// TIA Portal project "Takt_Docas_V13_SP1_V15" (V15)
// Software para a implementação do  Takt nas docas da fábrica do "KD".

(* hardware
DEVICE "S7-1200 station_1"  S7-1200 Station
   slot 0: "Rack_0"  Rack  V1.0
   slot 1: "PLC_Docas"  CPU 1214C DC/DC/DC  6ES7 214-1AG40-0XB0  V4.0
*)

// ===== PLC "PLC_Docas"  CPU 1214C DC/DC/DC =====

VAR_GLOBAL   // PLC tag table "Default tag table"
   "System_Byte" AT %MB1 : Byte;
   "FirstScan" AT %M1.0 : Bool;
   "DiagStatusUpdate" AT %M1.1 : Bool;
   "AlwaysTRUE" AT %M1.2 : Bool;
   "AlwaysFALSE" AT %M1.3 : Bool;
   "Clock_Byte" AT %MB0 : Byte;
   "Clock_10Hz" AT %M0.0 : Bool;
   "Clock_5Hz" AT %M0.1 : Bool;
   "Clock_2.5Hz" AT %M0.2 : Bool;
   "Clock_2Hz" AT %M0.3 : Bool;
   "Clock_1.25Hz" AT %M0.4 : Bool;
   "Clock_1Hz" AT %M0.5 : Bool;
   "Clock_0.625Hz" AT %M0.6 : Bool;
   "Clock_0.5Hz" AT %M0.7 : Bool;
   "Tag_1" AT %M100.0 : Bool;
   "startsystem" AT %I1.0 : Bool;
END_VAR

VAR_GLOBAL   // PLC tag table "Peripheral_inputs"
   "P.IN_Reset_Andon_doca1" AT %I0.0 : Bool;   // Entrada pereférica para resetar a chamada de Andon da "doca 1"
   "P.IN_Andon_doca1" AT %I0.1 : Bool;   // Entrada pereférica para chamada de Andon "doca 1"
   "P.IN_Reset_Andon_doca2" AT %I0.2 : Bool;   // Entrada pereférica para resetar a chamada de Andon da "doca 2"
   "P.IN_Andon_doca2" AT %I0.3 : Bool;   // Entrada pereférica para chamada de Andon "doca 2"
   "P.IN_Reset_Andon_doca3" AT %I0.4 : Bool;   // Entrada pereférica para resetar a chamada de Andon da "doca 3"
   "P.IN_Andon_doca3" AT %I0.5 : Bool;   // Entrada pereférica para chamada de Andon "doca 3"
   "P.IN_Reset_Andon_doca4" AT %I0.6 : Bool;   // Entrada pereférica para resetar a chamada de Andon da "doca 4"
   "P.IN_Andon_doca4" AT %I0.7 : Bool;   // Entrada pereférica para chamada de Andon "doca 4"
END_VAR

// folder: DBs

DATA_BLOCK "Input_memory"   // DB1
{ S7_Optimized_Access := 'TRUE' }
VERSION : 0.1
   VAR
      "M.S_IN_Reset_Andon_doca1" : Bool;   // Memória de movimentação do sinal de entrada do reset da chamada de Andon "doca1".
      "M.S_IN_Andon_doca1" : Bool;   // Memória de movimentação do sinal de entrada para chamada de andon "doca1".
      "M.S_IN_Reset_Andon_doca2" : Bool;   // Memória de movimentação do sinal de entrada do reset da chamada de Andon "doca2".
      "M.S_IN_Andon_doca2" : Bool;   // Memória de movimentação do sinal de entrada para chamada de andon "doca2".
      "M.S_IN_Reset_Andon_doca3" : Bool;   // Memória de movimentação do sinal de entrada do reset da chamada de Andon "doca3".
      "M.S_IN_Andon_doca3" : Bool;   // Memória de movimentação do sinal de entrada para chamada de andon "doca3".
      "M.S_IN_Reset_Andon_doca4" : Bool;   // Memória de movimentação do sinal de entrada do reset da chamada de Andon "doca4".
      "M.S_IN_Andon_doca4" : Bool;   // Memória de movimentação do sinal de entrada para chamada de andon "doca4".
   END_VAR
BEGIN
END_DATA_BLOCK

DATA_BLOCK "Output_memory"   // DB2
{ S7_Optimized_Access := 'TRUE' }
VERSION : 0.1
BEGIN
END_DATA_BLOCK

// folder: DBs_FBs

DATA_BLOCK "FB500_Dock_Takt_DB"   // DB3
{ S7_Optimized_Access := 'FALSE' }
VERSION : 0.1
// stored: InstanceOfName FB500_Dock_Takt
"FB500_Dock_Takt"
BEGIN
END_DATA_BLOCK

DATA_BLOCK "FB500_Dock_Takt_DB_1"   // DB4
{ S7_Optimized_Access := 'FALSE' }
VERSION : 0.1
// stored: InstanceOfName FB500_Dock_Takt
"FB500_Dock_Takt"
BEGIN
END_DATA_BLOCK

DATA_BLOCK "FB500_Dock_Takt_DB_2"   // DB5
{ S7_Optimized_Access := 'FALSE' }
VERSION : 0.1
// stored: InstanceOfName FB500_Dock_Takt
"FB500_Dock_Takt"
BEGIN
END_DATA_BLOCK

DATA_BLOCK "FB500_Dock_Takt_DB_3"   // DB6
{ S7_Optimized_Access := 'FALSE' }
VERSION : 0.1
// stored: InstanceOfName FB500_Dock_Takt
"FB500_Dock_Takt"
BEGIN
END_DATA_BLOCK

DATA_BLOCK "stopstar_DB"   // DB9
{ S7_Optimized_Access := 'TRUE' }
VERSION : 0.1
// stored: InstanceOfName Andon_Call
"Andon_Call"
BEGIN
END_DATA_BLOCK

// folder: DBs_System

DATA_BLOCK "Inputs_memory.system"   // DB7
{ S7_Optimized_Access := 'FALSE' }
VERSION : 0.1
   VAR
      "M.S_IN_Timer.Takt.D1" : Time;   // Memória de leitura do Sistema para parâmetrizar o tempo do Takt na "doca 1".
      "M.S_IN_Dock_goal.D1" : Int;   // Memória de leitura do Sistema para parâmetrizar o objetivo de produção na "doca 1".
      "M.S_IN_Timer.Takt.D2" : Time;   // Memória de leitura do Sistema para parâmetrizar o tempo do Takt na "doca 2".
      "M.S_IN_Dock_goal.D2" : Int;   // Memória de leitura do Sistema para parâmetrizar o objetivo de produção na "doca 2".
      "M.S_IN_Timer.Takt.D3" : Time;   // Memória de leitura do Sistema para parâmetrizar o tempo do Takt na "doca 3".
      "M.S_IN_Dock_goal.D3" : Int;   // Memória de leitura do Sistema para parâmetrizar o objetivo de produção na "doca 3".
      "M.S_IN_Timer.Takt.D4" : Time;   // Memória de leitura do Sistema para parâmetrizar o tempo do Takt na "doca 4".
      "M.S_IN_Dock_goal.D4" : Int;   // Memória de leitura do Sistema para parâmetrizar o objetivo de produção na "doca 4".
      "M.S_IN_Enable.Takt" : Bool;   // Memória de leitura do Sistema para habilitar o Takt das docas.
      StartBySystem1 : Bool;
      StartBySystem2 : Bool;
      StartBySystem3 : Bool;
      StartBySystem4 : Bool;
      Empty5 : Bool;
      Empty6 : Bool;
      Empty7 : Bool;
   END_VAR
BEGIN
END_DATA_BLOCK

DATA_BLOCK "Outputs_memory.system"   // DB8
{ S7_Optimized_Access := 'FALSE' }
VERSION : 0.1
   VAR
      "M.S_Out_TaktActual.D1" : Time;   // Memória de leitura do Sistema com o valor do Takt atual da "doca 1".
      "M.S_Out_StopTime.D1" : Time;   // Memória de leitura do Sistema com o valor do Stop time da "doca 1".
      "M.S_Out_Production.D1" : Int;   // Memória de leitura do Sistema com o valor da Produção até o momento da "doca 1"
      "M.S_Out_Dock_goal.D1" : Int;   // Memória de leitura do Sistema com o valor do objetivo de produção da "doca 1"
      "M.S_Out_TaktActual.D2" : Time;   // Memória de leitura do Sistema com o valor do Takt atual da "doca 2".
      "M.S_Out_StopTime.D2" : Time;   // Memória de leitura do Sistema com o valor do Stop time da "doca 2".
      "M.S_Out_Production.D2" : Int;   // Memória de leitura do Sistema com o valor da Produção até o momento da "doca 2"
      "M.S_Out_Dock_goal.D2" : Int;   // Memória de leitura do Sistema com o valor do objetivo de produção da "doca 2"
      "M.S_Out_TaktActual.D3" : Time;   // Memória de leitura do Sistema com o valor do Takt atual da "doca 3".
      "M.S_Out_StopTime.D3" : Time;   // Memória de leitura do Sistema com o valor do Stop time da "doca 3".
      "M.S_Out_Production.D3" : Int;   // Memória de leitura do Sistema com o valor da Produção até o momento da "doca 3"
      "M.S_Out_Dock_goal.D3" : Int;   // Memória de leitura do Sistema com o valor do objetivo de produção da "doca 3"
      "M.S_Out_TaktActual.D4" : Time;   // Memória de leitura do Sistema com o valor do Takt atual da "doca 4".
      "M.S_Out_StopTime.D4" : Time;   // Memória de leitura do Sistema com o valor do Stop time da "doca 4".
      "M.S_Out_Production.D4" : Int;   // Memória de leitura do Sistema com o valor da Produção até o momento da "doca 4"
      "M.S_Out_Dock_goal.D4" : Int;   // Memória de leitura do Sistema com o valor do objetivo de produção da "doca 4"
      "M.S_Out_Stuffing_target" : Int;   // Memória de leitura do Sistema com o valor do objetivo diario total da estufagem.
      "M.S_Out_Andon.D1" : Bool;   // Memória de leitura do Sistema da chamada de Andon da "doca 1".
      "M.S_Out_Andon.D2" : Bool;   // Memória de leitura do Sistema da chamada de Andon da "doca 2".
      "M.S_Out_Andon.D3" : Bool;   // Memória de leitura do Sistema da chamada de Andon da "doca 3".
      "M.S_Out_Andon.D4" : Bool;   // Memória de leitura do Sistema da chamada de Andon da "doca 4".
      Empty : Bool;
      Empty_1 : Bool;
      Empty_2 : Bool;
      Empty_3 : Bool;
   END_VAR
BEGIN
END_DATA_BLOCK

// folder: (top level)

ORGANIZATION_BLOCK "Main"   // OB1, LAD, ProgramCycle
TITLE = "Main Program Sweep (Cycle)"
{ S7_Optimized_Access := 'TRUE' }
VERSION : 0.1
   VAR_INPUT
      Initial_Call : Bool;   // Initial call of this OB
      Remanence : Bool;   // =True, if remanent data are available
   END_VAR
BEGIN

REGION Network 1: Peripheral Signals (Andon_Call)
   // Movimentação dos sinais das entradas periféricas para as memórias de movimentação.
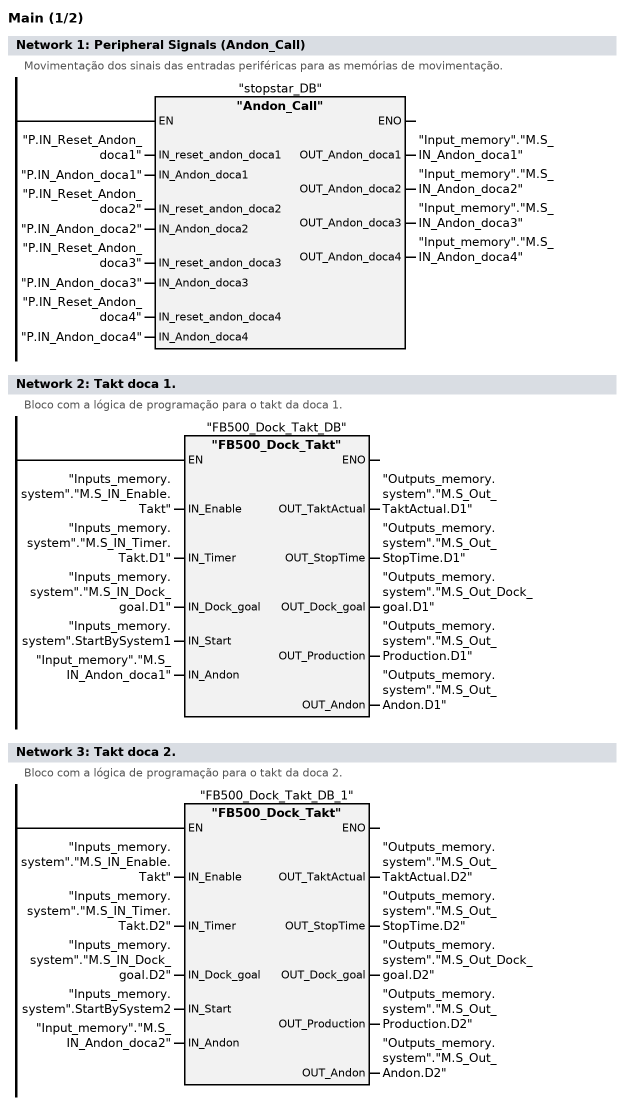
   RUNG wire#powerrail
      "stopstar_DB"(IN_reset_andon_doca1 := "P.IN_Reset_Andon_doca1", IN_Andon_doca1 := "P.IN_Andon_doca1", IN_reset_andon_doca2 := "P.IN_Reset_Andon_doca2", IN_Andon_doca2 := "P.IN_Andon_doca2", IN_reset_andon_doca3 := "P.IN_Reset_Andon_doca3", IN_Andon_doca3 := "P.IN_Andon_doca3", IN_reset_andon_doca4 := "P.IN_Reset_Andon_doca4", IN_Andon_doca4 := "P.IN_Andon_doca4", OUT_Andon_doca1 => "Input_memory"."M.S_IN_Andon_doca1", OUT_Andon_doca2 => "Input_memory"."M.S_IN_Andon_doca2", OUT_Andon_doca3 => "Input_memory"."M.S_IN_Andon_doca3", OUT_Andon_doca4 => "Input_memory"."M.S_IN_Andon_doca4")
   END_RUNG
   // the same network as SCL:
   "stopstar_DB"(IN_reset_andon_doca1 := "P.IN_Reset_Andon_doca1",   // "Andon_Call"
                 IN_Andon_doca1 := "P.IN_Andon_doca1",
                 IN_reset_andon_doca2 := "P.IN_Reset_Andon_doca2",
                 IN_Andon_doca2 := "P.IN_Andon_doca2",
                 IN_reset_andon_doca3 := "P.IN_Reset_Andon_doca3",
                 IN_Andon_doca3 := "P.IN_Andon_doca3",
                 IN_reset_andon_doca4 := "P.IN_Reset_Andon_doca4",
                 IN_Andon_doca4 := "P.IN_Andon_doca4",
                 OUT_Andon_doca1 => "Input_memory"."M.S_IN_Andon_doca1",
                 OUT_Andon_doca2 => "Input_memory"."M.S_IN_Andon_doca2",
                 OUT_Andon_doca3 => "Input_memory"."M.S_IN_Andon_doca3",
                 OUT_Andon_doca4 => "Input_memory"."M.S_IN_Andon_doca4");
END_REGION

REGION Network 2: Takt doca 1.
   // Bloco com a lógica de programação para o takt da doca 1.
   RUNG wire#powerrail
      "FB500_Dock_Takt_DB"(IN_Enable := "Inputs_memory.system"."M.S_IN_Enable.Takt", IN_Timer := "Inputs_memory.system"."M.S_IN_Timer.Takt.D1", IN_Dock_goal := "Inputs_memory.system"."M.S_IN_Dock_goal.D1", IN_Start := "Inputs_memory.system".StartBySystem1, IN_Andon := "Input_memory"."M.S_IN_Andon_doca1", OUT_TaktActual => "Outputs_memory.system"."M.S_Out_TaktActual.D1", OUT_StopTime => "Outputs_memory.system"."M.S_Out_StopTime.D1", OUT_Dock_goal => "Outputs_memory.system"."M.S_Out_Dock_goal.D1", OUT_Production => "Outputs_memory.system"."M.S_Out_Production.D1", OUT_Andon => "Outputs_memory.system"."M.S_Out_Andon.D1")
   END_RUNG
   // the same network as SCL:
   "FB500_Dock_Takt_DB"(IN_Enable := "Inputs_memory.system"."M.S_IN_Enable.Takt",   // "FB500_Dock_Takt"
                        IN_Timer := "Inputs_memory.system"."M.S_IN_Timer.Takt.D1",
                        IN_Dock_goal := "Inputs_memory.system"."M.S_IN_Dock_goal.D1",
                        IN_Start := "Inputs_memory.system".StartBySystem1,
                        IN_Andon := "Input_memory"."M.S_IN_Andon_doca1",
                        OUT_TaktActual => "Outputs_memory.system"."M.S_Out_TaktActual.D1",
                        OUT_StopTime => "Outputs_memory.system"."M.S_Out_StopTime.D1",
                        OUT_Dock_goal => "Outputs_memory.system"."M.S_Out_Dock_goal.D1",
                        OUT_Production => "Outputs_memory.system"."M.S_Out_Production.D1",
                        OUT_Andon => "Outputs_memory.system"."M.S_Out_Andon.D1");
END_REGION

REGION Network 3: Takt doca 2.
   // Bloco com a lógica de programação para o takt da doca 2.
   RUNG wire#powerrail
      "FB500_Dock_Takt_DB_1"(IN_Enable := "Inputs_memory.system"."M.S_IN_Enable.Takt", IN_Timer := "Inputs_memory.system"."M.S_IN_Timer.Takt.D2", IN_Dock_goal := "Inputs_memory.system"."M.S_IN_Dock_goal.D2", IN_Start := "Inputs_memory.system".StartBySystem2, IN_Andon := "Input_memory"."M.S_IN_Andon_doca2", OUT_TaktActual => "Outputs_memory.system"."M.S_Out_TaktActual.D2", OUT_StopTime => "Outputs_memory.system"."M.S_Out_StopTime.D2", OUT_Dock_goal => "Outputs_memory.system"."M.S_Out_Dock_goal.D2", OUT_Production => "Outputs_memory.system"."M.S_Out_Production.D2", OUT_Andon => "Outputs_memory.system"."M.S_Out_Andon.D2")
   END_RUNG
   // the same network as SCL:
   "FB500_Dock_Takt_DB_1"(IN_Enable := "Inputs_memory.system"."M.S_IN_Enable.Takt",   // "FB500_Dock_Takt"
                          IN_Timer := "Inputs_memory.system"."M.S_IN_Timer.Takt.D2",
                          IN_Dock_goal := "Inputs_memory.system"."M.S_IN_Dock_goal.D2",
                          IN_Start := "Inputs_memory.system".StartBySystem2,
                          IN_Andon := "Input_memory"."M.S_IN_Andon_doca2",
                          OUT_TaktActual => "Outputs_memory.system"."M.S_Out_TaktActual.D2",
                          OUT_StopTime => "Outputs_memory.system"."M.S_Out_StopTime.D2",
                          OUT_Dock_goal => "Outputs_memory.system"."M.S_Out_Dock_goal.D2",
                          OUT_Production => "Outputs_memory.system"."M.S_Out_Production.D2",
                          OUT_Andon => "Outputs_memory.system"."M.S_Out_Andon.D2");
END_REGION

REGION Network 4: Takt doca 3.
   // Bloco com a lógica de programação para o takt da doca 3.
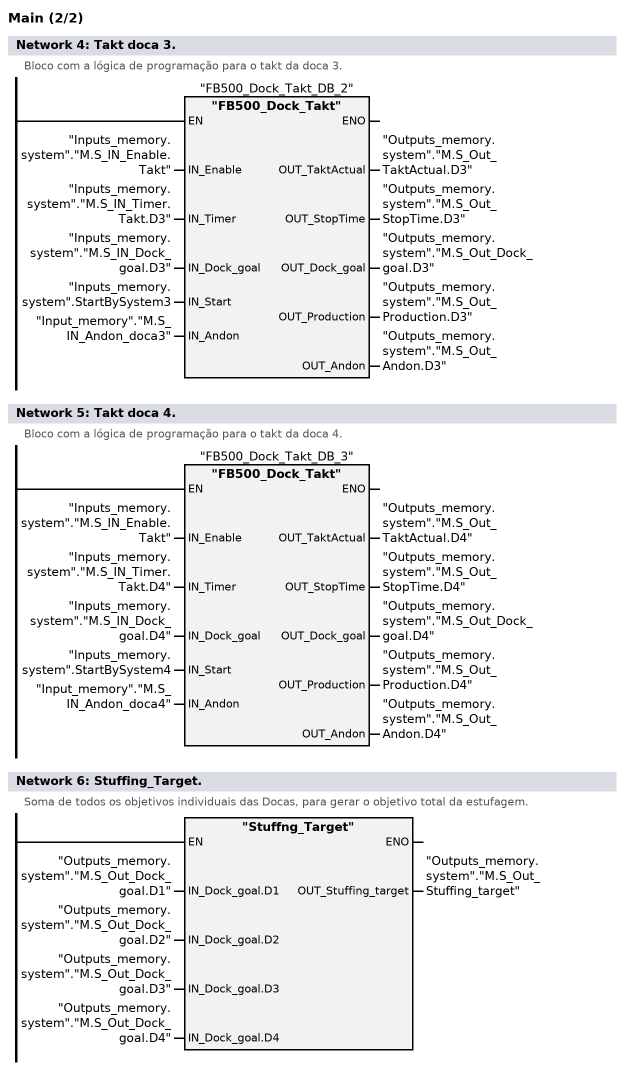
   RUNG wire#powerrail
      "FB500_Dock_Takt_DB_2"(IN_Enable := "Inputs_memory.system"."M.S_IN_Enable.Takt", IN_Timer := "Inputs_memory.system"."M.S_IN_Timer.Takt.D3", IN_Dock_goal := "Inputs_memory.system"."M.S_IN_Dock_goal.D3", IN_Start := "Inputs_memory.system".StartBySystem3, IN_Andon := "Input_memory"."M.S_IN_Andon_doca3", OUT_TaktActual => "Outputs_memory.system"."M.S_Out_TaktActual.D3", OUT_StopTime => "Outputs_memory.system"."M.S_Out_StopTime.D3", OUT_Dock_goal => "Outputs_memory.system"."M.S_Out_Dock_goal.D3", OUT_Production => "Outputs_memory.system"."M.S_Out_Production.D3", OUT_Andon => "Outputs_memory.system"."M.S_Out_Andon.D3")
   END_RUNG
   // the same network as SCL:
   "FB500_Dock_Takt_DB_2"(IN_Enable := "Inputs_memory.system"."M.S_IN_Enable.Takt",   // "FB500_Dock_Takt"
                          IN_Timer := "Inputs_memory.system"."M.S_IN_Timer.Takt.D3",
                          IN_Dock_goal := "Inputs_memory.system"."M.S_IN_Dock_goal.D3",
                          IN_Start := "Inputs_memory.system".StartBySystem3,
                          IN_Andon := "Input_memory"."M.S_IN_Andon_doca3",
                          OUT_TaktActual => "Outputs_memory.system"."M.S_Out_TaktActual.D3",
                          OUT_StopTime => "Outputs_memory.system"."M.S_Out_StopTime.D3",
                          OUT_Dock_goal => "Outputs_memory.system"."M.S_Out_Dock_goal.D3",
                          OUT_Production => "Outputs_memory.system"."M.S_Out_Production.D3",
                          OUT_Andon => "Outputs_memory.system"."M.S_Out_Andon.D3");
END_REGION

REGION Network 5: Takt doca 4.
   // Bloco com a lógica de programação para o takt da doca 4.
   RUNG wire#powerrail
      "FB500_Dock_Takt_DB_3"(IN_Enable := "Inputs_memory.system"."M.S_IN_Enable.Takt", IN_Timer := "Inputs_memory.system"."M.S_IN_Timer.Takt.D4", IN_Dock_goal := "Inputs_memory.system"."M.S_IN_Dock_goal.D4", IN_Start := "Inputs_memory.system".StartBySystem4, IN_Andon := "Input_memory"."M.S_IN_Andon_doca4", OUT_TaktActual => "Outputs_memory.system"."M.S_Out_TaktActual.D4", OUT_StopTime => "Outputs_memory.system"."M.S_Out_StopTime.D4", OUT_Dock_goal => "Outputs_memory.system"."M.S_Out_Dock_goal.D4", OUT_Production => "Outputs_memory.system"."M.S_Out_Production.D4", OUT_Andon => "Outputs_memory.system"."M.S_Out_Andon.D4")
   END_RUNG
   // the same network as SCL:
   "FB500_Dock_Takt_DB_3"(IN_Enable := "Inputs_memory.system"."M.S_IN_Enable.Takt",   // "FB500_Dock_Takt"
                          IN_Timer := "Inputs_memory.system"."M.S_IN_Timer.Takt.D4",
                          IN_Dock_goal := "Inputs_memory.system"."M.S_IN_Dock_goal.D4",
                          IN_Start := "Inputs_memory.system".StartBySystem4,
                          IN_Andon := "Input_memory"."M.S_IN_Andon_doca4",
                          OUT_TaktActual => "Outputs_memory.system"."M.S_Out_TaktActual.D4",
                          OUT_StopTime => "Outputs_memory.system"."M.S_Out_StopTime.D4",
                          OUT_Dock_goal => "Outputs_memory.system"."M.S_Out_Dock_goal.D4",
                          OUT_Production => "Outputs_memory.system"."M.S_Out_Production.D4",
                          OUT_Andon => "Outputs_memory.system"."M.S_Out_Andon.D4");
END_REGION

REGION Network 6: Stuffing_Target.
   // Soma de todos os objetivos individuais das Docas, para gerar o objetivo total da estufagem.
   RUNG wire#powerrail
      "Stuffng_Target"("IN_Dock_goal.D1" := "Outputs_memory.system"."M.S_Out_Dock_goal.D1", "IN_Dock_goal.D2" := "Outputs_memory.system"."M.S_Out_Dock_goal.D2", "IN_Dock_goal.D3" := "Outputs_memory.system"."M.S_Out_Dock_goal.D3", "IN_Dock_goal.D4" := "Outputs_memory.system"."M.S_Out_Dock_goal.D4", OUT_Stuffing_target => "Outputs_memory.system"."M.S_Out_Stuffing_target")
   END_RUNG
   // the same network as SCL:
   "Stuffng_Target"("IN_Dock_goal.D1" := "Outputs_memory.system"."M.S_Out_Dock_goal.D1",
                    "IN_Dock_goal.D2" := "Outputs_memory.system"."M.S_Out_Dock_goal.D2",
                    "IN_Dock_goal.D3" := "Outputs_memory.system"."M.S_Out_Dock_goal.D3",
                    "IN_Dock_goal.D4" := "Outputs_memory.system"."M.S_Out_Dock_goal.D4",
                    OUT_Stuffing_target => "Outputs_memory.system"."M.S_Out_Stuffing_target");
END_REGION
END_ORGANIZATION_BLOCK

// folder: FBs

FUNCTION_BLOCK "FB500_Dock_Takt"   // FB1, SCL
{ S7_Optimized_Access := 'FALSE' }
VERSION : 0.1
   VAR_INPUT
      IN_Enable : Bool;   // Sinal para habilitação do takt.
      IN_Timer : Time;   // Regulagem do tempo contado pelo takt.
      IN_Dock_goal : Int;   // Sinal de parametrização do objetivo de produção individual da doca.
      IN_Start : Bool;   // Sinal para inicio de contagem do tempo de takt.
      IN_Andon : Bool;   // Sinal para chamada de ajuda.
   END_VAR
   VAR_OUTPUT
      OUT_TaktActual : Time;   // Tempo do takt.
      OUT_StopTime : Time;   // Tempo de Stop time.
      OUT_Dock_goal : Int;   // Objetivo de produção individual da doca.
      OUT_Production : Int;   // Produção até o momento.
      OUT_Andon : Bool;   // Chamada de ajuda (Andon).
   END_VAR
   VAR
      S_TaktTimer : TON_TIME;   // Temporizador para o takt.
      S_StopTime_Timer : TON_TIME;   // Temporizador para o Stop time.
      "S_Timer.PT" : Time;   // "Preset time" do temporizador do takt.
      "S_Timer.ET" : Time;   // "Elapsed Time" do temporizador do takt.
      "S_Timer2.ET" : Time;   // "Elapsed Time" do temporizador do Stop time.
      "S_Timer.IN" : Bool;   // "Start" do temporizador do takt.
      "S_Timer_Takt.Q" : Bool;   // "Output" do temporizador do takt.
      S_Pulse : Bool;   // Pulso de pausa do temporizador do takt.
      S_Pulse2 : Bool;   // Pulso de pausa do temporizador do Stop time.
      S_PulseFlag : Bool;   // Pulso Auxiliar de pausa do temporizador do takt.
      S_PulseFlag2 : Bool;   // Pulso Auxiliar de pausa do temporizador do Stop time.
      "S_Accum.Time" : Time;   // Acumula o tempo do temporizador do Takt quando foi pausado.
      "S_AccumTime.Stop" : Time;   // Acumula o tempo do temporizador do Stop time quando foi pausado.
      S_Sequence : Int;   // Sequencia para execução da lógica.
      S_StopTime : Time;   // Auxiliar tempo de Stop time.
      S_TaktActual : Time;   // Auxiliar tempo do takt.
      "S_Timer.IN_2" : Bool;   // "Start" do temporizador do Stop time.
      S_Counter : CTU_INT;   // Production Counter
      S_CounterValue : Int;   // Contador para atribuir o valor de produção até o momento.
      S_CounterReset : Bool;   // "Reset" para o contador de produção até o momento.
      S_Andon : Bool;   // Auxiliar chamada de ajuda (Andon).
   END_VAR
BEGIN

   //INITIAL ROUTINE
   IF #IN_Enable AND #S_Sequence = 0 THEN

       #S_StopTime := T#0s;
       #"S_AccumTime.Stop" := T#0s;
       #S_TaktActual := #IN_Timer;
       #"S_Accum.Time" := T#0s;
       #"S_Timer.PT" := #IN_Timer;
       #"S_Timer.ET" := T#0s;
       #"S_Timer2.ET" := T#0s;
       #"S_Timer.IN_2" := 0;
       #S_CounterReset := 1;
       #OUT_Dock_goal := #IN_Dock_goal;
       #S_Sequence := 1;
   END_IF;

   //TAKT ROUTINE
   IF #IN_Enable AND #S_Sequence = 1 THEN

       //START (TAKT TIME) TIMER. 
       IF #IN_Start AND
           NOT #IN_Andon THEN

           #"S_Timer.IN" := 1;

       END_IF;

       //_________________________________________________________________________________________________________________________________________________

       //STOP TIMER TAKT.

       IF #"S_Timer_Takt.Q" THEN
           #"S_Timer.IN" := 0;

       END_IF;


       //_________________________________________________________________________________________________________________________________________________

       //PULSE GENERATE TAKT.

       #S_Pulse := NOT #"S_Timer.IN" AND #S_PulseFlag;
       #S_PulseFlag := #"S_Timer.IN";

       //_________________________________________________________________________________________________________________________________________________

       IF #S_Pulse THEN

           #"S_Accum.Time" := #"S_Timer.ET";
           #"S_Timer.PT" := #"S_Timer.PT" - #"S_Accum.Time";

       END_IF;

       //_________________________________________________________________________________________________________________________________________________

       // ACTUAL TAKT.

       #S_TaktActual := #"S_Timer.PT" - #"S_Timer.ET";
       #OUT_TaktActual := #S_TaktActual;

       //_________________________________________________________________________________________________________________________________________________  

       // RESET VALUES AT THE END OF TAKT. 
       IF #"S_Timer_Takt.Q" THEN

           #"S_Accum.Time" := T#0s;
           #"S_Timer.PT" := #IN_Timer;
           #"S_Timer.ET" := T#0s;
           #S_TaktActual := #IN_Timer;

       END_IF;
       //_________________________________________________________________________________________________________________________________________________   

       // START FOR THE ANDON CALL.

           #S_Andon := #IN_Andon;


       // CALL OF ANDON IN DOCA.

       #OUT_Andon := #S_Andon;

       IF #"S_Timer_Takt.Q" AND #S_Andon THEN
           #"S_Timer.IN_2" := 1;

       END_IF;

       //_________________________________________________________________________________________________________________________________________________    

       // RESET STOP TIMER/ ANDON.

       IF NOT #S_Andon THEN
           #"S_Timer.IN_2" := 0;

       END_IF;
       //_________________________________________________________________________________________________________________________________________________ 

       //PULSE_2 GENERATE STOP TIME.

       #S_Pulse2 := NOT #"S_Timer.IN_2" AND #S_PulseFlag2;
       #S_PulseFlag2 := #"S_Timer.IN_2";
       //_________________________________________________________________________________________________________________________________________________ 

       IF #S_Pulse2 THEN
           #"S_AccumTime.Stop" := #"S_Timer2.ET" + #"S_AccumTime.Stop";

       END_IF;
       //_________________________________________________________________________________________________________________________________________________ 

       #S_StopTime := #"S_AccumTime.Stop" + #"S_Timer2.ET";
       #OUT_StopTime := #S_StopTime;

   END_IF;

   // TIMER TAKT.

   #S_TaktTimer(IN := #"S_Timer.IN",
                PT := #"S_Timer.PT",
                Q => #"S_Timer_Takt.Q",
                ET => #"S_Timer.ET");

   // TIMER STOP TIME.
   #S_StopTime_Timer(IN := #"S_Timer.IN_2",
                     PT := T#9h,
                     ET => #"S_Timer2.ET");

   //PRODUCTION COUNTER.
   IF #"S_Timer.PT" > t#1s THEN
       #S_Counter(CU := #S_TaktTimer.Q,
                  CV => #S_CounterValue,
                  PV := 999,
                  R := #S_CounterReset);
   END_IF;

   #S_CounterReset := 0;
   #OUT_Production := #S_CounterValue;

   //END ROUTINE.
   IF NOT #IN_Enable THEN

       #S_Sequence := 0;
       #"S_Timer.IN" := 0;

   END_IF;
END_FUNCTION_BLOCK

FUNCTION_BLOCK "Andon_Call"   // FB2, SCL
{ S7_Optimized_Access := 'TRUE' }
VERSION : 0.1
   VAR_INPUT
      IN_reset_andon_doca1 : Bool;   // Sinal de entrada periférica para reset andon "doca 1".
      IN_Andon_doca1 : Bool;   // Sinal de entrada periférica para chamada de andon "doca 1".
      IN_reset_andon_doca2 : Bool;   // Sinal de entrada periférica para reset andon "doca 2".
      IN_Andon_doca2 : Bool;   // Sinal de entrada periférica para chamada de andon "doca 2".
      IN_reset_andon_doca3 : Bool;   // Sinal de entrada periférica para reset andon "doca 3".
      IN_Andon_doca3 : Bool;   // Sinal de entrada periférica para chamada de andon "doca 3".
      IN_reset_andon_doca4 : Bool;   // Sinal de entrada periférica para reset andon "doca 4".
      IN_Andon_doca4 : Bool;   // Sinal de entrada periférica para chamada de andon "doca 4".
   END_VAR
   VAR_OUTPUT
      OUT_Andon_doca1 : Bool;   // Sinal para memória de movimentação da chamada de Andon da "doca1".
      OUT_Andon_doca2 : Bool;   // Sinal para memória de movimentação da chamada de Andon da "doca2".
      OUT_Andon_doca3 : Bool;   // Sinal para memória de movimentação da chamada de Andon da "doca3".
      OUT_Andon_doca4 : Bool;   // Sinal para memória de movimentação da chamada de Andon da "doca4".
   END_VAR
   VAR
      S_reset_andon_doca1 : Bool;   // Auxiliar para reset da chamada de andon "doca 1".
      S_Andon_doca1 : Bool;   // Auxiliar para chamada de andon "doca 1".
      S_reset_andon_doca2 : Bool;   // Auxiliar para reset da chamada de andon "doca 2".
      S_Andon_doca2 : Bool;   // Auxiliar para chamada de andon "doca 2".
      S_reset_andon_doca3 : Bool;   // Auxiliar para reset da chamada de andon "doca 3".
      S_Andon_doca3 : Bool;   // Auxiliar para chamada de andon "doca 3".
      S_reset_andon_doca4 : Bool;   // Auxiliar para reset da chamada de andon "doca 4".
      S_Andon_doca4 : Bool;   // Auxiliar para chamada de andon "doca 4".
      S_Andon_doca1_out : Bool;   // Auxiliar sinal de chamada de andon "verdade/falso" "doca 1"
      S_Andon_doca2_out : Bool;   // Auxiliar sinal de chamada de andon "verdade/falso" "doca 2"
      S_Andon_doca3_out : Bool;   // Auxiliar sinal de chamada de andon "verdade/falso" "doca 3"
      S_Andon_doca4_out : Bool;   // Auxiliar sinal de chamada de andon "verdade/falso" "doca 4"
   END_VAR
BEGIN
   // Movimentação dos sinais das entradas periféricas para as memórias de movimentação.

   #S_reset_andon_doca1 := #IN_reset_andon_doca1;
   #S_reset_andon_doca2 := #IN_reset_andon_doca2;
   #S_reset_andon_doca3 := #IN_reset_andon_doca3;
   #S_reset_andon_doca4 := #IN_reset_andon_doca4;
   #S_Andon_doca1 := #IN_Andon_doca1;
   #S_Andon_doca2 := #IN_Andon_doca2;
   #S_Andon_doca3 := #IN_Andon_doca3;
   #S_Andon_doca4 := #IN_Andon_doca4;

   // "Doca 1".

   IF #S_Andon_doca1  THEN
       #S_Andon_doca1_out := 1;
   END_IF;
   IF #S_reset_andon_doca1 THEN
       #S_Andon_doca1_out := 0;
   END_IF;

   //___________________________________________________________________________________________________________________________________________________________________________________________________________________

   // "Doca 2".
   IF #S_Andon_doca2 THEN
       #S_Andon_doca2_out := 1;
   END_IF;
   IF #S_reset_andon_doca2 THEN
       #S_Andon_doca2_out := 0;
   END_IF;

   //___________________________________________________________________________________________________________________________________________________________________________________________________________________

   // "Doca 3".
   IF #S_Andon_doca3 THEN
       #S_Andon_doca3_out := 1;
   END_IF;
   IF #S_reset_andon_doca3 THEN
       #S_Andon_doca3_out := 0;
   END_IF;

   //___________________________________________________________________________________________________________________________________________________________________________________________________________________

   // "Doca 4".
   IF #S_Andon_doca4 THEN
       #S_Andon_doca4_out := 1;
   END_IF;
   IF #S_reset_andon_doca4 THEN
       #S_Andon_doca4_out := 0;
   END_IF;

   //Output (Andon Call)
   #OUT_Andon_doca1 := #S_Andon_doca1_out;
   #OUT_Andon_doca2 := #S_Andon_doca2_out;
   #OUT_Andon_doca3 := #S_Andon_doca3_out;
   #OUT_Andon_doca4 := #S_Andon_doca4_out;
   //_______________________________________________________________________________________________________________________________________________________________________________________________________________
END_FUNCTION_BLOCK

// folder: FCs

FUNCTION "Stuffng_Target" : Void   // FC2, SCL
{ S7_Optimized_Access := 'TRUE' }
VERSION : 0.1
   VAR_INPUT
      "IN_Dock_goal.D1" : Int;   // Sinal da memória de leitura do Sistema com o valor do objetivo de produção da "doca 1".
      "IN_Dock_goal.D2" : Int;   // Sinal da memória de leitura do Sistema com o valor do objetivo de produção da "doca 2".
      "IN_Dock_goal.D3" : Int;   // Sinal da memória de leitura do Sistema com o valor do objetivo de produção da "doca 3".
      "IN_Dock_goal.D4" : Int;   // Sinal da memória de leitura do Sistema com o valor do objetivo de produção da "doca 4".
   END_VAR
   VAR_OUTPUT
      OUT_Stuffing_target : Int;   // Objetivo diario total da estufagem.
   END_VAR
BEGIN
   // Sum of individual dock targets.

   #OUT_Stuffing_target := #"IN_Dock_goal.D1" + #"IN_Dock_goal.D2" + #"IN_Dock_goal.D3" + #"IN_Dock_goal.D4";
END_FUNCTION